(* CoDeSys 2.3 export: FTURNOFFK14PUMP.EXP *)

(* POU fTurnOffK14Pump, ST *)
FUNCTION fTurnOffK14Pump : BOOL
VAR_INPUT
	PumpID : USINT;
END_VAR
VAR
END_VAR
	fSetK14Pump(FALSE, PumpID);
END_FUNCTION
